FUNCTION_BLOCK FB_SwitchableDecoratorBase IMPLEMENTS I_Switchable
VAR_INPUT
END_VAR
VAR_OUTPUT
END_VAR
VAR
	iSwitchable : I_Switchable;
END_VAR

PROPERTY Active : BOOL
GET
END_GET
END_PROPERTY

METHOD FB_init : BOOL
VAR_INPUT
	bInitRetains : BOOL; // if TRUE, the retain variables are initialized (warm start / cold start)
	bInCopyCode : BOOL;  // if TRUE, the instance afterwards gets moved into the copy code (online change)
	iSwitchable : I_Switchable; // The switchable to be decorated.
END_VAR
this^.iSwitchable := iSwitchable;
END_METHOD

METHOD Off : BOOL
END_METHOD

METHOD On : BOOL
END_METHOD

PROPERTY PUBLIC Switchable : BOOL
GET
Switchable := THIS^.iSwitchable;
END_GET
SET
THIS^.iSwitchable := Switchable;
END_SET
END_PROPERTY

END_FUNCTION_BLOCK

(* stored: Version 1.1.0.1, ProductVersion 3.1.4024.5
   POU FB_SwitchableDecoratorBase: Id {646ed8f0-9f88-4c29-b1cc-39ed1daea851}, SpecialFunc None
   Property Active: Id {2d0c3ea1-8442-4501-a287-61f937cba039}
   Get Get: Id {a6352963-d33b-4e55-8790-9750d031777b}
   Method FB_init: Id {22bb49a7-c28f-4f46-bafc-cf098b4ebe1e}
   Method Off: Id {1453815f-27d4-4370-9774-22a67bad95f2}
   Method On: Id {218a2d49-ee4c-405f-8b58-1c3db5bf7f78}
   Property Switchable: Id {642bef93-2d32-4d80-8746-c11d0387045f}
   Get Get: Id {2437e1b6-0d10-4898-ab36-9ce65545dd4f}
   Set Set: Id {80cb6a94-9e35-4421-940f-555484877df8} *)
